{attribute 'linkalways'} 
{attribute 'no_explicit_call' := 'This FB is a CLASS and must be accessed using methods or properties'}
{attribute 'enable_dynamic_creation'}
FUNCTION_BLOCK Node_F_VN_SetAt_TcVnRotatedRectangle EXTENDS VisionNode
VAR
    stElement : _TcVnRotatedRectangle;
    ipContainer : _ITcVnContainer;
    nIndex : _ULINT(0);
    hrPrev : _HRESULT(S_OK);
    hresult : _HRESULT(S_OK);
END_VAR

METHOD PUBLIC  Clone : I_Node
VAR
	pNode : POINTER TO Node_F_VN_SetAt_TcVnRotatedRectangle;
END_VAR
pNode := __NEW(Node_F_VN_SetAt_TcVnRotatedRectangle);
Clone := pNode^;
END_METHOD

METHOD FB_init : BOOL
VAR_INPUT
	bInitRetains : BOOL; // if TRUE, the retain variables are initialized (warm start / cold start)
	bInCopyCode : BOOL;  // if TRUE, the instance afterwards gets moved into the copy code (online change)
END_VAR
AddInput('stElement', stElement);
AddInput('ipContainer', ipContainer);
AddParameter('nIndex', nIndex);
AddInput('hrPrev', hrPrev);
AddOutput('ipContainer', ipContainer);
AddOutput('hresult',hresult);
END_METHOD

METHOD PROTECTED OnExecute
hresult.Value := F_VN_SetAt_TcVnRotatedRectangle(
    stElement := stElement.Value,
    ipContainer := ipContainer.Value,
    nIndex := nIndex.Value,
    hrPrev:= hrPrev.Value);
END_METHOD

METHOD PUBLIC PreExecutionCheck
VAR_INPUT
	Check : I_PreExecutionChecks;
END_VAR
Check.IsTrue(ipContainer.IsValid, 'ipContainer must be a valid container');
Check.IsTrue(ipContainer.HasType(TC_GLOBAL_CONST_LIST.ContainerType_Vector_TcVnRotatedRectangle), 'ipContainer contains incorrect type');
END_METHOD

END_FUNCTION_BLOCK

(* stored: Version 1.1.0.1, ProductVersion 3.1.4024.15
   POU Node_F_VN_SetAt_TcVnRotatedRectangle: Id {e3c59804-8c12-081b-2a79-86dd5484348a}, SpecialFunc None
   Folder Constructor: Id {80710085-4d47-0e93-3ef3-9e3cedd17058}
   Method Clone: Id {c8465e60-5234-017a-0f23-d33f4386f3f7}
   Method FB_init: Id {86b8b004-2395-0601-14c0-4510e574f903}
   Method OnExecute: Id {81b9d821-fe41-0640-3648-1a12e668e6fd}
   Method PreExecutionCheck: Id {0dde3891-3c41-0ccb-1c66-6a9ce1a8dab1} *)
